{attribute 'linkalways'} 
{attribute 'no_explicit_call' := 'This FB is a CLASS and must be accessed using methods or properties'}
{attribute 'enable_dynamic_creation'}
FUNCTION_BLOCK Node_F_VN_ConnectedComponentsWithStatsExp EXTENDS VisionNode
VAR
    ipSrcImage : _ITcVnImage;
    ipLabelImage : _ITcVnImage;
    ipBoundingBoxes : _ITcVnContainer;
    ipNumPixels : _ITcVnContainer;
    ipCentroids : _ITcVnContainer;
    nLabels : _DINT(0);
    eConnectivity : _ETcVnPixelConnectivity(ETcVnPixelConnectivity.TCVN_PC_4);
    eLabelType : _ETcVnElementType(ETcVnElementType.TCVN_ET_DINT);
    eAlgorithm : _ETcVnConnectedComponentsAlgorithm(ETcVnConnectedComponentsAlgorithm.TCVN_CCA_WU);
    hrPrev : _HRESULT(S_OK);
	hresult : _HRESULT(S_OK);
END_VAR

METHOD PUBLIC  Clone : I_Node
VAR
	pNode : POINTER TO Node_F_VN_ConnectedComponentsWithStatsExp;
END_VAR
pNode := __NEW(Node_F_VN_ConnectedComponentsWithStatsExp);
Clone := pNode^;
END_METHOD

METHOD FB_init : BOOL
VAR_INPUT
	bInitRetains : BOOL; // if TRUE, the retain variables are initialized (warm start / cold start)
	bInCopyCode : BOOL;  // if TRUE, the instance afterwards gets moved into the copy code (online change)
END_VAR
AddInput('ipSrcImage', ipSrcImage);
AddParameter('eConnectivity', eConnectivity);
AddParameter('eLabelType', eLabelType);
AddParameter('eAlgorithm', eAlgorithm);
AddInput('hrPrev', hrPrev);
AddOutput('ipLabelImage', ipLabelImage);
AddOutput('nLabels', nLabels);
AddOutput('hresult', hresult);
END_METHOD

METHOD PROTECTED OnExecute
hresult.Value := F_VN_ConnectedComponentsWithStatsExp(
	ipSrcImage := ipSrcImage.Value,
    ipLabelImage := ipLabelImage.Value,
    ipBoundingBoxes := ipBoundingBoxes.Value,
    ipNumPixels := ipNumPixels.Value,
    ipCentroids := ipCentroids.Value,
    nLabels := nLabels.Value,
    eConnectivity := eConnectivity.Value,
    eLabelType := eLabelType.Value,
    eAlgorithm := eAlgorithm.Value,
	hrPrev:= hrPrev.Value);
END_METHOD

METHOD PUBLIC PreExecutionCheck
VAR_INPUT
	Check : I_PreExecutionChecks;
END_VAR
Check.IsTrue(ipSrcImage.IsValid, 'ipSrcImage must contain an image');
Check.IsTrue(ipSrcImage.IsPixelDepth(8), 'ipSrcImage must be 8 bit pixel depth');
Check.IsTrue(ipSrcImage.HasChannelCount(1), 'ipSrcImage must contain 1 channel');
Check.IsTrue((eLabelType.Value = ETcVnElementType.TCVN_ET_DINT) OR
             (eLabelType.Value = ETcVnElementType.TCVN_ET_UINT), 'eLabelType must be DINT or UINT');
END_METHOD

END_FUNCTION_BLOCK

(* stored: Version 1.1.0.1, ProductVersion 3.1.4024.15
   POU Node_F_VN_ConnectedComponentsWithStatsExp: Id {64bbfe25-5095-04e4-2acd-afceaaef3e31}, SpecialFunc None
   Folder Constructor: Id {e13b5330-07c6-0d36-2d3e-1a0ddbacba27}
   Method Clone: Id {4d31e326-486e-0445-172c-b57b0532dd75}
   Method FB_init: Id {dba99416-d0aa-08f4-2521-881a8ec541e5}
   Method OnExecute: Id {187fde92-2ca9-0a09-3cf6-643be711da57}
   Method PreExecutionCheck: Id {7af31468-7b8b-0cda-2d80-c65332ff4919} *)
